{attribute 'pack_mode' := '1'}
    {attribute 'OPC.UA.DA' := '1'}
    {attribute 'OPC.UA.DA.StructuredType' := '1'}
    (*
    ST_RW_KW_Device_Info_Generic_HMI_IgnitionExp
    ==================================================
    Generated from Ignition UDT: RW_KW_Device_Info_Generic
    Total tags: 8
    Generated on: 2025-09-16 12:06:03
    *)
    TYPE ST_RW_KW_Device_Info_Generic_HMI_IgnitionExp :
    STRUCT
        {attribute 'OPC.UA.DA' := '1'}
        {attribute 'OPC.UA.DA.Access' := '1'}
        KW_Device_Error : BOOL := FALSE;		// Read-only tag
        {attribute 'OPC.UA.DA' := '1'}
        {attribute 'OPC.UA.DA.Access' := '1'}
        KW_Device_ScanRateMs : DINT := 0;		// Read-only tag
        {attribute 'OPC.UA.DA' := '1'}
        {attribute 'OPC.UA.DA.Access' := '1'}
        KW_Device_Enabled : BOOL := FALSE;		// Read-only tag
        {attribute 'OPC.UA.DA' := '1'}
        {attribute 'OPC.UA.DA.Access' := '1'}
        KW_Device_Description : STRING := '';		// Read-only tag
        {attribute 'OPC.UA.DA' := '1'}
        {attribute 'OPC.UA.DA.Access' := '1'}
        KW_Device_ActiveTagCount : DINT := 0;		// Read-only tag

        {attribute 'OPC.UA.DA' := '1'}
        {attribute 'OPC.UA.DA.Access' := '1'}
        KW_Device_SecondsInError : SINT := 0;		// Read-only tag
        {attribute 'OPC.UA.DA' := '1'}
        {attribute 'OPC.UA.DA.Access' := '1'}
        IPAddress : STRING := '';		// Read-only tag
        {attribute 'OPC.UA.DA' := '1'}
        {attribute 'OPC.UA.DA.Access' := '1'}
        KW_Device_ScanMode : STRING := '';		// Read-only tag
    END_STRUCT
    END_TYPE

(* stored: Version 1.1.0.1
   DUT ST_RW_KW_Device_Info_Generic_HMI_IgnitionExp: Id {c26178b5-b008-4a3c-9250-daf9aab9c5da} *)
